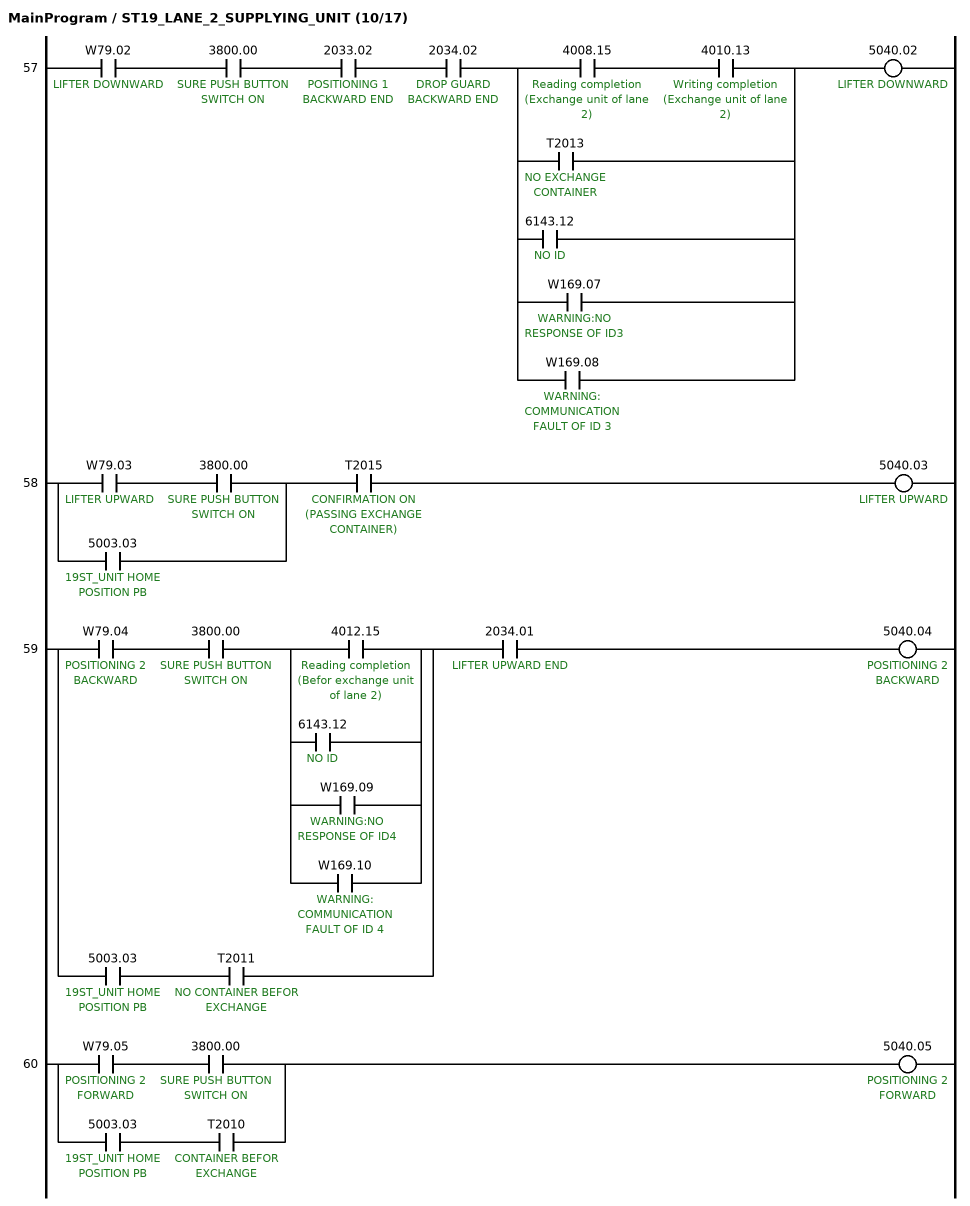
; [picture p696: MainProgram / ST19_LANE_2_SUPPLYING_UNIT, rungs 57-60]
; rung 57
LD W79.02  ; LIFTER DOWNWARD
AND 3800.00  ; SURE PUSH BUTTON SWITCH ON
AND 2033.02  ; POSITIONING 1 BACKWARD END
AND 2034.02  ; DROP GUARD BACKWARD END
LD 4008.15  ; Reading completion (Exchange unit of lane 2)
AND 4010.13  ; Writing completion (Exchange unit of lane 2)
OR T2013  ; NO EXCHANGE CONTAINER
OR 6143.12  ; NO ID
OR W169.07  ; WARNING:NO RESPONSE OF ID3
OR W169.08  ; WARNING:COMMUNICATION FAULT OF ID 3
ANDLD
OUT 5040.02  ; LIFTER DOWNWARD
; rung 58
LD W79.03  ; LIFTER UPWARD
AND 3800.00  ; SURE PUSH BUTTON SWITCH ON
OR 5003.03  ; 19ST_UNIT HOME POSITION PB
AND T2015  ; CONFIRMATION ON (PASSING EXCHANGE CONTAINER)
OUT 5040.03  ; LIFTER UPWARD
; rung 59
LD W79.04  ; POSITIONING 2 BACKWARD
AND 3800.00  ; SURE PUSH BUTTON SWITCH ON
LD 4012.15  ; Reading completion (Befor exchange unit of lane 2)
OR 6143.12  ; NO ID
OR W169.09  ; WARNING:NO RESPONSE OF ID4
OR W169.10  ; WARNING:COMMUNICATION FAULT OF ID 4
ANDLD
LD 5003.03  ; 19ST_UNIT HOME POSITION PB
AND T2011  ; NO CONTAINER BEFOR EXCHANGE
ORLD
AND 2034.01  ; LIFTER UPWARD END
OUT 5040.04  ; POSITIONING 2 BACKWARD
; rung 60
LD W79.05  ; POSITIONING 2 FORWARD
AND 3800.00  ; SURE PUSH BUTTON SWITCH ON
LD 5003.03  ; 19ST_UNIT HOME POSITION PB
AND T2010  ; CONTAINER BEFOR EXCHANGE
ORLD
OUT 5040.05  ; POSITIONING 2 FORWARD

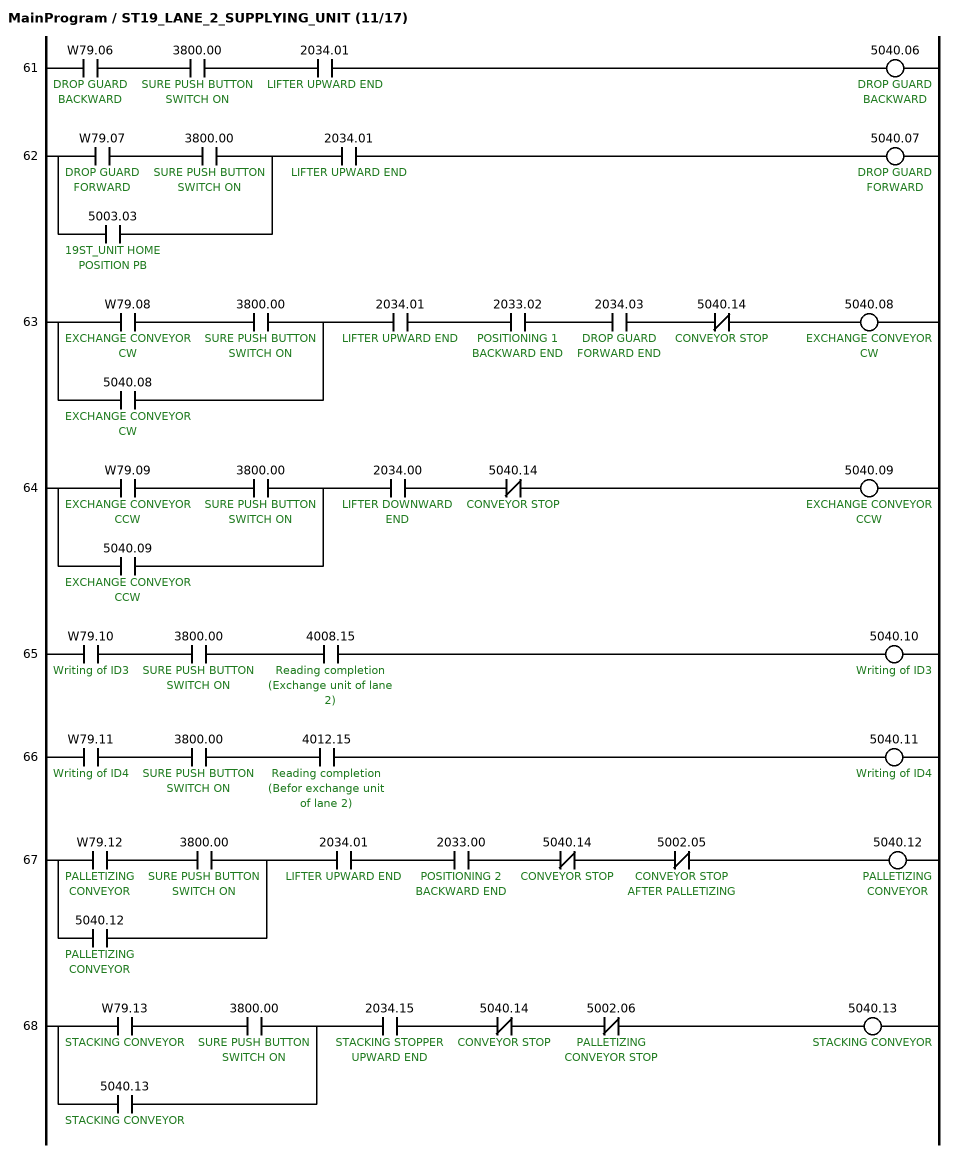
; rung 61
LD W79.06  ; DROP GUARD BACKWARD
AND 3800.00  ; SURE PUSH BUTTON SWITCH ON
AND 2034.01  ; LIFTER UPWARD END
OUT 5040.06  ; DROP GUARD BACKWARD
; rung 62
LD W79.07  ; DROP GUARD FORWARD
AND 3800.00  ; SURE PUSH BUTTON SWITCH ON
OR 5003.03  ; 19ST_UNIT HOME POSITION PB
AND 2034.01  ; LIFTER UPWARD END
OUT 5040.07  ; DROP GUARD FORWARD
; rung 63
LD W79.08  ; EXCHANGE CONVEYOR CW
AND 3800.00  ; SURE PUSH BUTTON SWITCH ON
OR 5040.08  ; EXCHANGE CONVEYOR CW
AND 2034.01  ; LIFTER UPWARD END
AND 2033.02  ; POSITIONING 1 BACKWARD END
AND 2034.03  ; DROP GUARD FORWARD END
ANDNOT 5040.14  ; CONVEYOR STOP
OUT 5040.08  ; EXCHANGE CONVEYOR CW
; rung 64
LD W79.09  ; EXCHANGE CONVEYOR CCW
AND 3800.00  ; SURE PUSH BUTTON SWITCH ON
OR 5040.09  ; EXCHANGE CONVEYOR CCW
AND 2034.00  ; LIFTER DOWNWARD END
ANDNOT 5040.14  ; CONVEYOR STOP
OUT 5040.09  ; EXCHANGE CONVEYOR CCW
; rung 65
LD W79.10  ; Writing of ID3
AND 3800.00  ; SURE PUSH BUTTON SWITCH ON
AND 4008.15  ; Reading completion (Exchange unit of lane 2)
OUT 5040.10  ; Writing of ID3
; rung 66
LD W79.11  ; Writing of ID4
AND 3800.00  ; SURE PUSH BUTTON SWITCH ON
AND 4012.15  ; Reading completion (Befor exchange unit of lane 2)
OUT 5040.11  ; Writing of ID4
; rung 67
LD W79.12  ; PALLETIZING CONVEYOR
AND 3800.00  ; SURE PUSH BUTTON SWITCH ON
OR 5040.12  ; PALLETIZING CONVEYOR
AND 2034.01  ; LIFTER UPWARD END
AND 2033.00  ; POSITIONING 2 BACKWARD END
ANDNOT 5040.14  ; CONVEYOR STOP
ANDNOT 5002.05  ; CONVEYOR STOP AFTER PALLETIZING
OUT 5040.12  ; PALLETIZING CONVEYOR
; rung 68
LD W79.13  ; STACKING CONVEYOR
AND 3800.00  ; SURE PUSH BUTTON SWITCH ON
OR 5040.13  ; STACKING CONVEYOR
AND 2034.15  ; STACKING STOPPER UPWARD END
ANDNOT 5040.14  ; CONVEYOR STOP
ANDNOT 5002.06  ; PALLETIZING CONVEYOR STOP
OUT 5040.13  ; STACKING CONVEYOR

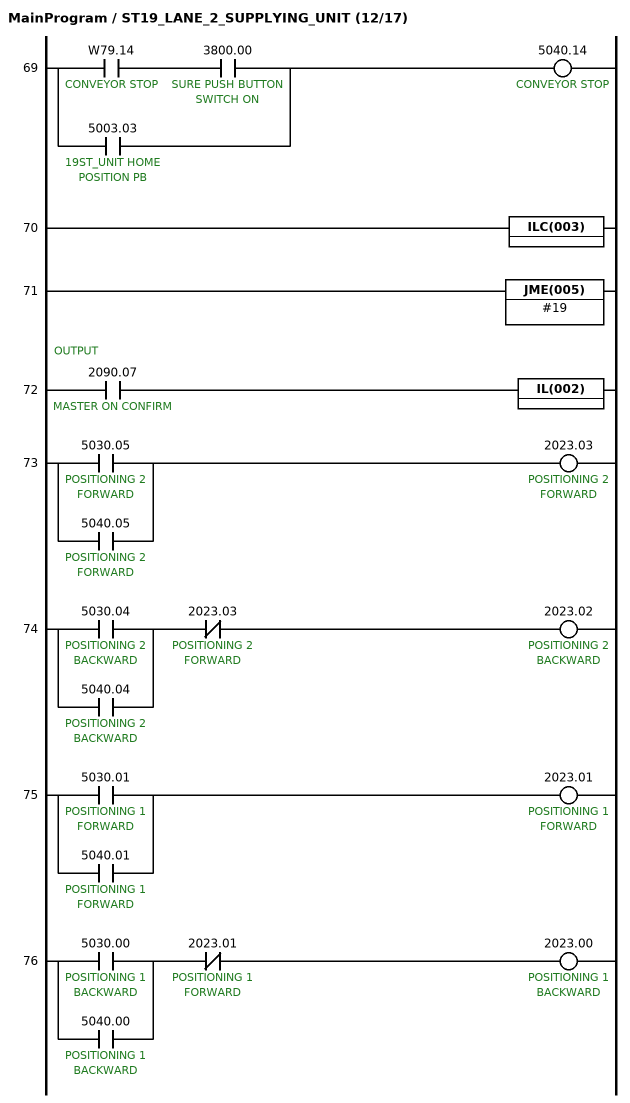
; rung 69
LD W79.14  ; CONVEYOR STOP
AND 3800.00  ; SURE PUSH BUTTON SWITCH ON
OR 5003.03  ; 19ST_UNIT HOME POSITION PB
OUT 5040.14  ; CONVEYOR STOP
; rung 70
ILC(003)
; rung 71
JME(005) #19
; rung 72: OUTPUT
LD 2090.07  ; MASTER ON CONFIRM
IL(002)
; rung 73
LD 5030.05  ; POSITIONING 2 FORWARD
OR 5040.05  ; POSITIONING 2 FORWARD
OUT 2023.03  ; POSITIONING 2 FORWARD
; rung 74
LD 5030.04  ; POSITIONING 2 BACKWARD
OR 5040.04  ; POSITIONING 2 BACKWARD
ANDNOT 2023.03  ; POSITIONING 2 FORWARD
OUT 2023.02  ; POSITIONING 2 BACKWARD
; rung 75
LD 5030.01  ; POSITIONING 1 FORWARD
OR 5040.01  ; POSITIONING 1 FORWARD
OUT 2023.01  ; POSITIONING 1 FORWARD
; rung 76
LD 5030.00  ; POSITIONING 1 BACKWARD
OR 5040.00  ; POSITIONING 1 BACKWARD
ANDNOT 2023.01  ; POSITIONING 1 FORWARD
OUT 2023.00  ; POSITIONING 1 BACKWARD

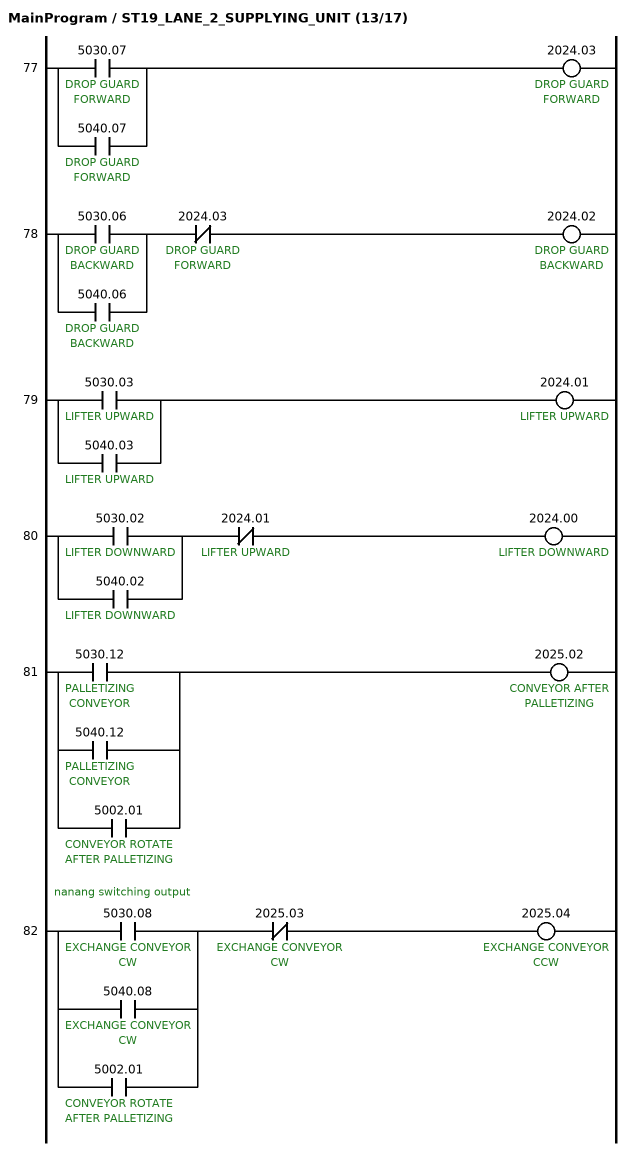
; rung 77
LD 5030.07  ; DROP GUARD FORWARD
OR 5040.07  ; DROP GUARD FORWARD
OUT 2024.03  ; DROP GUARD FORWARD
; rung 78
LD 5030.06  ; DROP GUARD BACKWARD
OR 5040.06  ; DROP GUARD BACKWARD
ANDNOT 2024.03  ; DROP GUARD FORWARD
OUT 2024.02  ; DROP GUARD BACKWARD
; rung 79
LD 5030.03  ; LIFTER UPWARD
OR 5040.03  ; LIFTER UPWARD
OUT 2024.01  ; LIFTER UPWARD
; rung 80
LD 5030.02  ; LIFTER DOWNWARD
OR 5040.02  ; LIFTER DOWNWARD
ANDNOT 2024.01  ; LIFTER UPWARD
OUT 2024.00  ; LIFTER DOWNWARD
; rung 81
LD 5030.12  ; PALLETIZING CONVEYOR
OR 5040.12  ; PALLETIZING CONVEYOR
OR 5002.01  ; CONVEYOR ROTATE AFTER PALLETIZING
OUT 2025.02  ; CONVEYOR AFTER PALLETIZING
; rung 82: nanang switching output
LD 5030.08  ; EXCHANGE CONVEYOR CW
OR 5040.08  ; EXCHANGE CONVEYOR CW
OR 5002.01  ; CONVEYOR ROTATE AFTER PALLETIZING
ANDNOT 2025.03  ; EXCHANGE CONVEYOR CW
OUT 2025.04  ; EXCHANGE CONVEYOR CCW

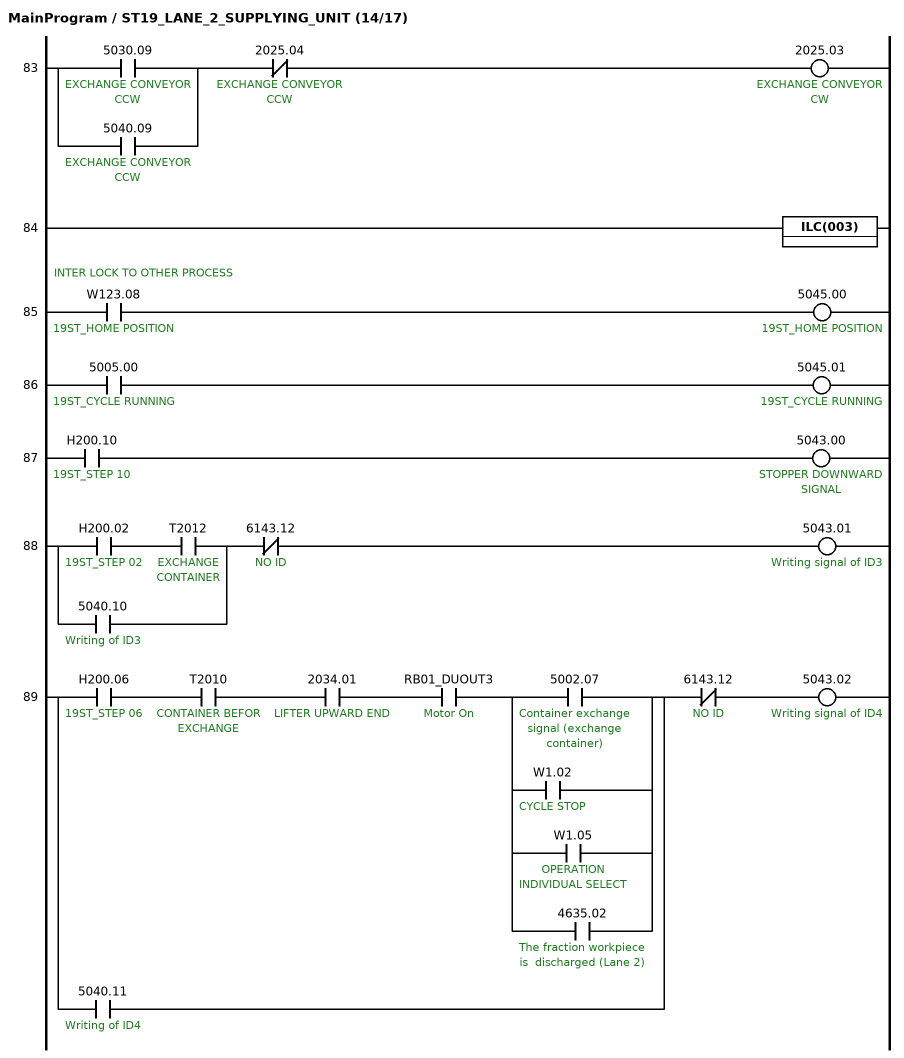
; rung 83
LD 5030.09  ; EXCHANGE CONVEYOR CCW
OR 5040.09  ; EXCHANGE CONVEYOR CCW
ANDNOT 2025.04  ; EXCHANGE CONVEYOR CCW
OUT 2025.03  ; EXCHANGE CONVEYOR CW
; rung 84
ILC(003)
; rung 85: INTER LOCK TO OTHER PROCESS
LD W123.08  ; 19ST_HOME POSITION
OUT 5045.00  ; 19ST_HOME POSITION
; rung 86
LD 5005.00  ; 19ST_CYCLE RUNNING
OUT 5045.01  ; 19ST_CYCLE RUNNING
; rung 87
LD H200.10  ; 19ST_STEP 10
OUT 5043.00  ; STOPPER DOWNWARD SIGNAL
; rung 88
LD H200.02  ; 19ST_STEP 02
AND T2012  ; EXCHANGE CONTAINER
OR 5040.10  ; Writing of ID3
ANDNOT 6143.12  ; NO ID
OUT 5043.01  ; Writing signal of ID3
; rung 89
LD H200.06  ; 19ST_STEP 06
AND T2010  ; CONTAINER BEFOR EXCHANGE
AND 2034.01  ; LIFTER UPWARD END
AND RB01_DUOUT3  ; Motor On
LD 5002.07  ; Container exchange signal (exchange container)
OR W1.02  ; CYCLE STOP
OR W1.05  ; OPERATION INDIVIDUAL SELECT
OR 4635.02  ; The fraction workpiece is  discharged (Lane 2)
ANDLD
OR 5040.11  ; Writing of ID4
ANDNOT 6143.12  ; NO ID
OUT 5043.02  ; Writing signal of ID4

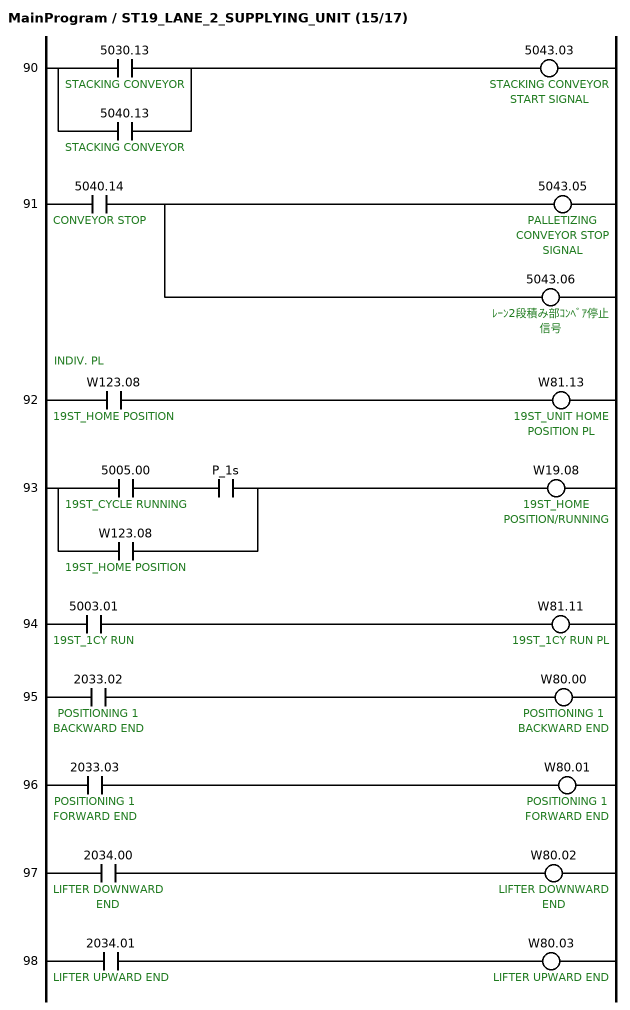
; rung 90
LD 5030.13  ; STACKING CONVEYOR
OR 5040.13  ; STACKING CONVEYOR
OUT 5043.03  ; STACKING CONVEYOR START SIGNAL
; rung 91
LD 5040.14  ; CONVEYOR STOP
OUT 5043.05  ; PALLETIZING CONVEYOR STOP SIGNAL
OUT 5043.06  ; ﾚｰﾝ2段積み部ｺﾝﾍﾞｱ停止信号
; rung 92: INDIV. PL
LD W123.08  ; 19ST_HOME POSITION
OUT W81.13  ; 19ST_UNIT HOME POSITION PL
; rung 93
LD 5005.00  ; 19ST_CYCLE RUNNING
AND P_1s
OR W123.08  ; 19ST_HOME POSITION
OUT W19.08  ; 19ST_HOME POSITION/RUNNING
; rung 94
LD 5003.01  ; 19ST_1CY RUN
OUT W81.11  ; 19ST_1CY RUN PL
; rung 95
LD 2033.02  ; POSITIONING 1 BACKWARD END
OUT W80.00  ; POSITIONING 1 BACKWARD END
; rung 96
LD 2033.03  ; POSITIONING 1 FORWARD END
OUT W80.01  ; POSITIONING 1 FORWARD END
; rung 97
LD 2034.00  ; LIFTER DOWNWARD END
OUT W80.02  ; LIFTER DOWNWARD END
; rung 98
LD 2034.01  ; LIFTER UPWARD END
OUT W80.03  ; LIFTER UPWARD END

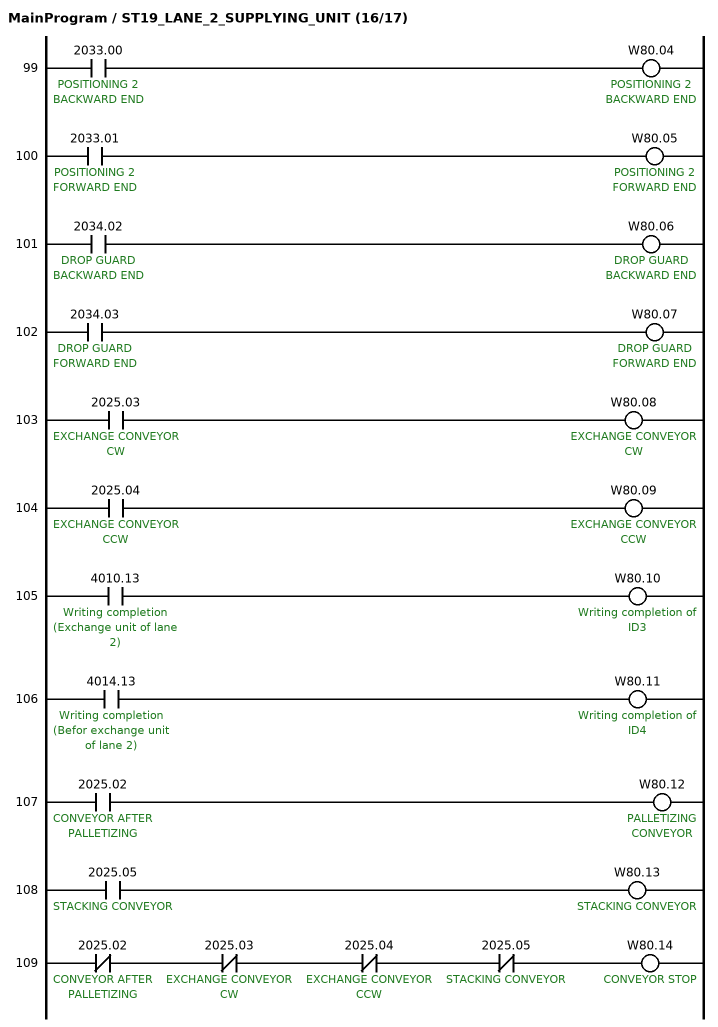
; rung 99
LD 2033.00  ; POSITIONING 2 BACKWARD END
OUT W80.04  ; POSITIONING 2 BACKWARD END
; rung 100
LD 2033.01  ; POSITIONING 2 FORWARD END
OUT W80.05  ; POSITIONING 2 FORWARD END
; rung 101
LD 2034.02  ; DROP GUARD BACKWARD END
OUT W80.06  ; DROP GUARD BACKWARD END
; rung 102
LD 2034.03  ; DROP GUARD FORWARD END
OUT W80.07  ; DROP GUARD FORWARD END
; rung 103
LD 2025.03  ; EXCHANGE CONVEYOR CW
OUT W80.08  ; EXCHANGE CONVEYOR CW
; rung 104
LD 2025.04  ; EXCHANGE CONVEYOR CCW
OUT W80.09  ; EXCHANGE CONVEYOR CCW
; rung 105
LD 4010.13  ; Writing completion (Exchange unit of lane 2)
OUT W80.10  ; Writing completion of ID3
; rung 106
LD 4014.13  ; Writing completion (Befor exchange unit of lane 2)
OUT W80.11  ; Writing completion of ID4
; rung 107
LD 2025.02  ; CONVEYOR AFTER PALLETIZING
OUT W80.12  ; PALLETIZING CONVEYOR
; rung 108
LD 2025.05  ; STACKING CONVEYOR
OUT W80.13  ; STACKING CONVEYOR
; rung 109
LDNOT 2025.02  ; CONVEYOR AFTER PALLETIZING
ANDNOT 2025.03  ; EXCHANGE CONVEYOR CW
ANDNOT 2025.04  ; EXCHANGE CONVEYOR CCW
ANDNOT 2025.05  ; STACKING CONVEYOR
OUT W80.14  ; CONVEYOR STOP

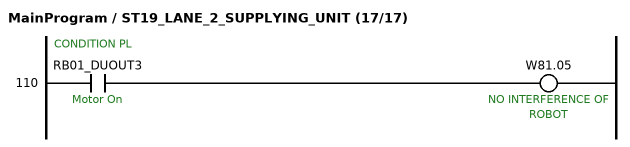
; rung 110: CONDITION PL
LD RB01_DUOUT3  ; Motor On
OUT W81.05  ; NO INTERFERENCE OF ROBOT

### Section ST20_LANE_2_STACKING_UNIT

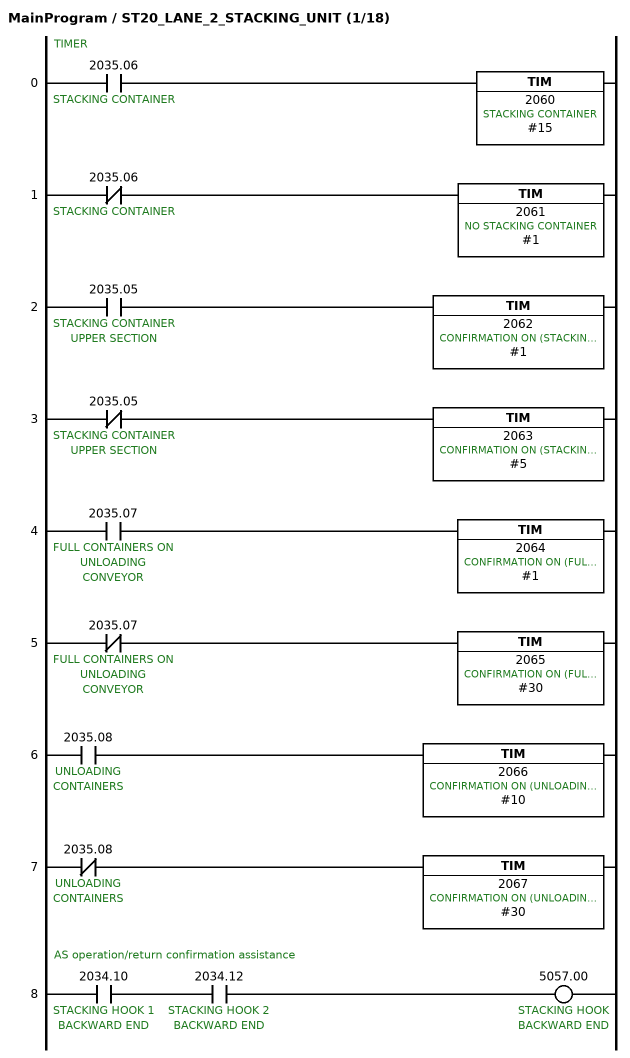
; rung 0: TIMER
LD 2035.06  ; STACKING CONTAINER
TIM 2060 #15  ; STACKING CONTAINER
; rung 1
LDNOT 2035.06  ; STACKING CONTAINER
TIM 2061 #1  ; NO STACKING CONTAINER
; rung 2
LD 2035.05  ; STACKING CONTAINER UPPER SECTION
TIM 2062 #1  ; CONFIRMATION ON (STACKING CONTAINER UPPER SECTION)
; rung 3
LDNOT 2035.05  ; STACKING CONTAINER UPPER SECTION
TIM 2063 #5  ; CONFIRMATION ON (STACKING CONTAINER UPPER SECTION)
; rung 4
LD 2035.07  ; FULL CONTAINERS ON UNLOADING CONVEYOR
TIM 2064 #1  ; CONFIRMATION ON (FULL CONTAINERS ON UNLOADING CONVEYOR)
; rung 5
LDNOT 2035.07  ; FULL CONTAINERS ON UNLOADING CONVEYOR
TIM 2065 #30  ; CONFIRMATION ON (FULL CONTAINERS ON UNLOADING CONVEYOR)
; rung 6
LD 2035.08  ; UNLOADING CONTAINERS
TIM 2066 #10  ; CONFIRMATION ON (UNLOADING CONTAINERS)
; rung 7
LDNOT 2035.08  ; UNLOADING CONTAINERS
TIM 2067 #30  ; CONFIRMATION ON (UNLOADING CONTAINERS)
; rung 8: AS operation/return confirmation assistance
LD 2034.10  ; STACKING HOOK 1 BACKWARD END
AND 2034.12  ; STACKING HOOK 2 BACKWARD END
OUT 5057.00  ; STACKING HOOK BACKWARD END

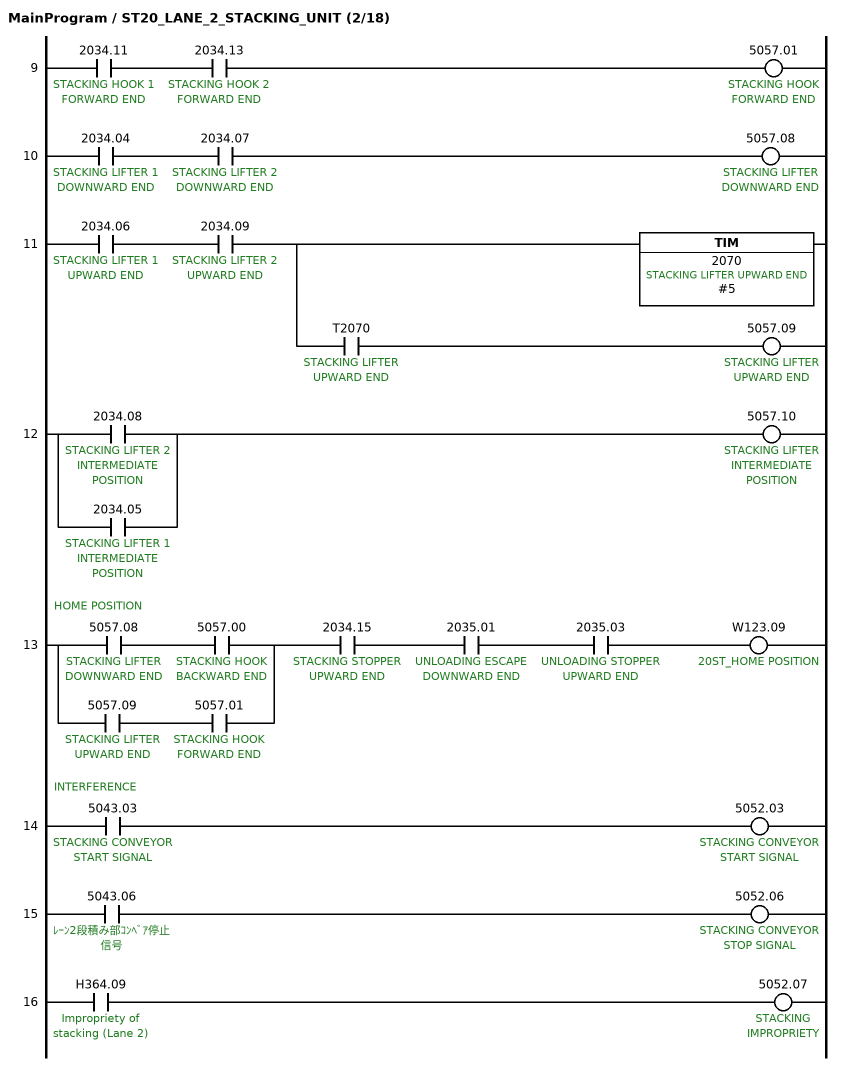
; rung 9
LD 2034.11  ; STACKING HOOK 1 FORWARD END
AND 2034.13  ; STACKING HOOK 2 FORWARD END
OUT 5057.01  ; STACKING HOOK FORWARD END
; rung 10
LD 2034.04  ; STACKING LIFTER 1 DOWNWARD END
AND 2034.07  ; STACKING LIFTER 2 DOWNWARD END
OUT 5057.08  ; STACKING LIFTER DOWNWARD END
; rung 11
LD 2034.06  ; STACKING LIFTER 1 UPWARD END
AND 2034.09  ; STACKING LIFTER 2 UPWARD END
TIM 2070 #5  ; STACKING LIFTER UPWARD END
AND T2070  ; STACKING LIFTER UPWARD END
OUT 5057.09  ; STACKING LIFTER UPWARD END
; rung 12
LD 2034.08  ; STACKING LIFTER 2 INTERMEDIATE POSITION
OR 2034.05  ; STACKING LIFTER 1 INTERMEDIATE POSITION
OUT 5057.10  ; STACKING LIFTER INTERMEDIATE POSITION
; rung 13: HOME POSITION
LD 5057.08  ; STACKING LIFTER DOWNWARD END
AND 5057.00  ; STACKING HOOK BACKWARD END
LD 5057.09  ; STACKING LIFTER UPWARD END
AND 5057.01  ; STACKING HOOK FORWARD END
ORLD
AND 2034.15  ; STACKING STOPPER UPWARD END
AND 2035.01  ; UNLOADING ESCAPE DOWNWARD END
AND 2035.03  ; UNLOADING STOPPER UPWARD END
OUT W123.09  ; 20ST_HOME POSITION
; rung 14: INTERFERENCE
LD 5043.03  ; STACKING CONVEYOR START SIGNAL
OUT 5052.03  ; STACKING CONVEYOR START SIGNAL
; rung 15
LD 5043.06  ; ﾚｰﾝ2段積み部ｺﾝﾍﾞｱ停止信号
OUT 5052.06  ; STACKING CONVEYOR STOP SIGNAL
; rung 16
LD H364.09  ; Impropriety of stacking (Lane 2)
OUT 5052.07  ; STACKING IMPROPRIETY

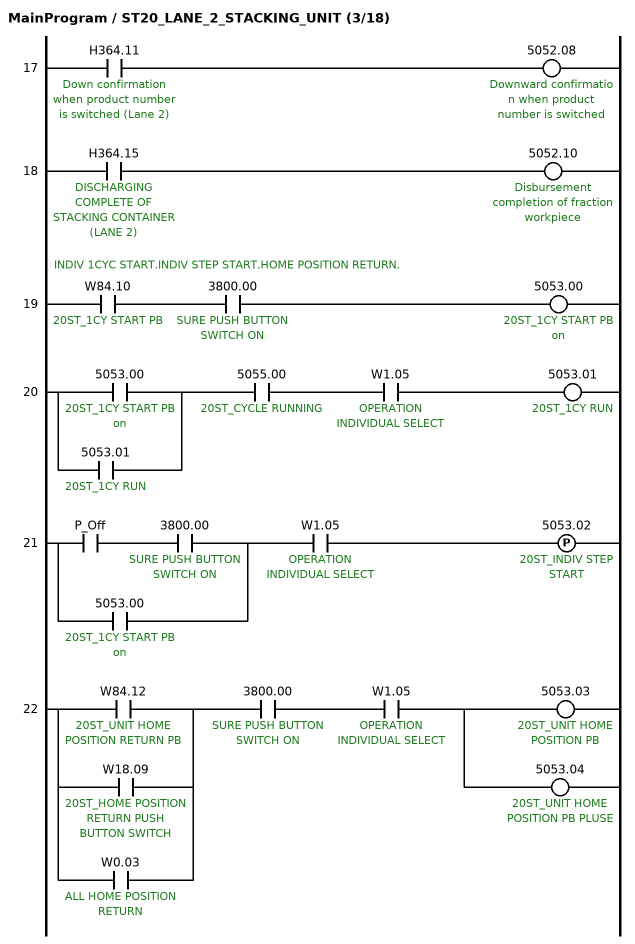
; rung 17
LD H364.11  ; Down confirmation when product number is switched (Lane 2)
OUT 5052.08  ; Downward confirmation when product number is switched
; rung 18
LD H364.15  ; DISCHARGING COMPLETE OF STACKING CONTAINER  (LANE 2)
OUT 5052.10  ; Disbursement completion of fraction workpiece
; rung 19: INDIV 1CYC START.INDIV STEP START.HOME POSITION RETURN.
LD W84.10  ; 20ST_1CY START PB
AND 3800.00  ; SURE PUSH BUTTON SWITCH ON
OUT 5053.00  ; 20ST_1CY START PB on
; rung 20
LD 5053.00  ; 20ST_1CY START PB on
OR 5053.01  ; 20ST_1CY RUN
AND 5055.00  ; 20ST_CYCLE RUNNING
AND W1.05  ; OPERATION INDIVIDUAL SELECT
OUT 5053.01  ; 20ST_1CY RUN
; rung 21
LD P_Off
AND 3800.00  ; SURE PUSH BUTTON SWITCH ON
OR 5053.00  ; 20ST_1CY START PB on
AND W1.05  ; OPERATION INDIVIDUAL SELECT
DIFU(013) 5053.02  ; 20ST_INDIV STEP START
; rung 22
LD W84.12  ; 20ST_UNIT HOME POSITION RETURN PB
OR W18.09  ; 20ST_HOME POSITION RETURN PUSH BUTTON SWITCH
OR W0.03  ; ALL HOME POSITION RETURN
AND 3800.00  ; SURE PUSH BUTTON SWITCH ON
AND W1.05  ; OPERATION INDIVIDUAL SELECT
OUT 5053.03  ; 20ST_UNIT HOME POSITION PB
OUT 5053.04  ; 20ST_UNIT HOME POSITION PB PLUSE

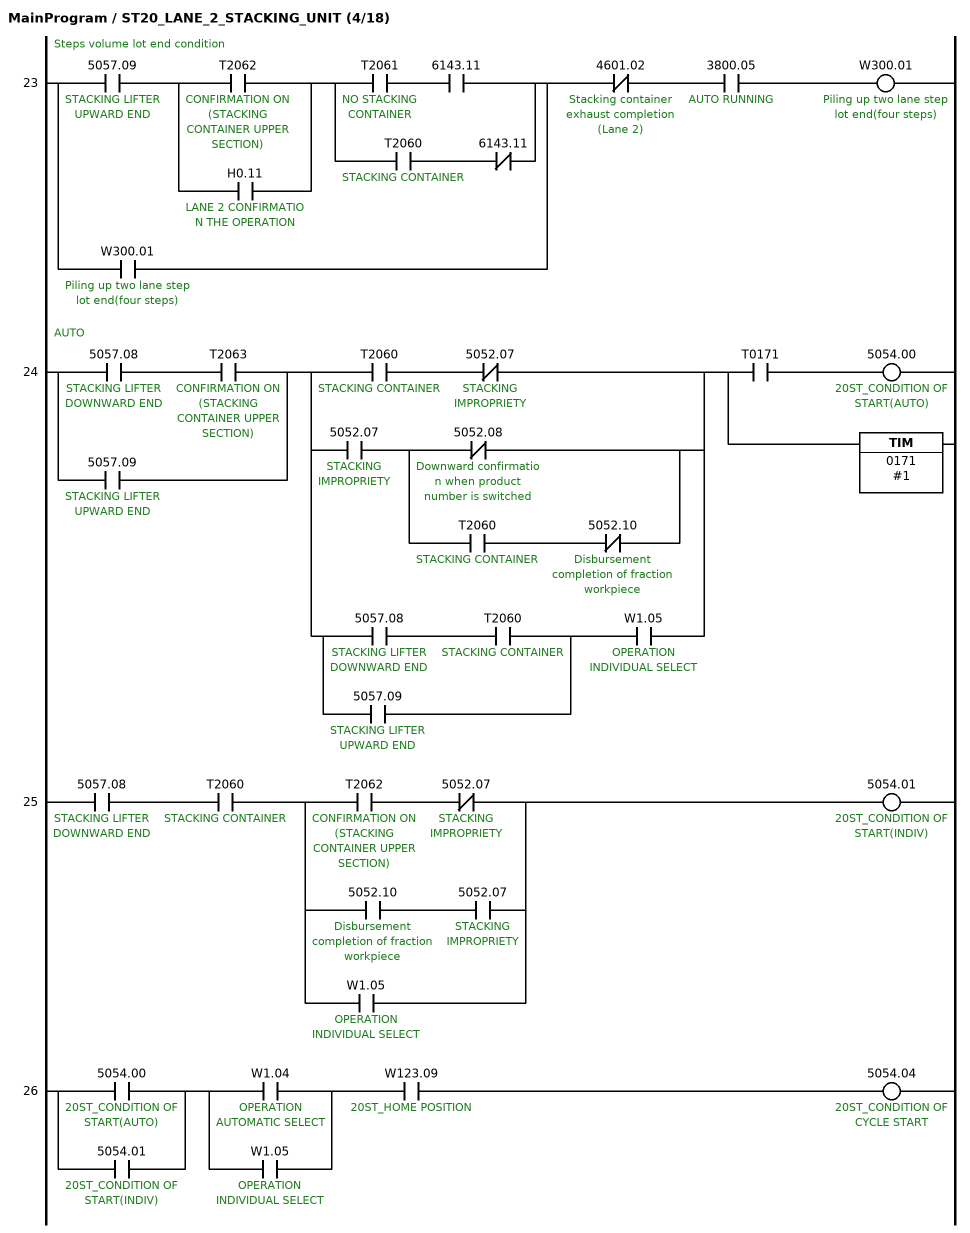
; rung 23: Steps volume lot end condition
LD 5057.09  ; STACKING LIFTER UPWARD END
LD T2062  ; CONFIRMATION ON (STACKING CONTAINER UPPER SECTION)
OR H0.11  ; LANE 2 CONFIRMATION THE OPERATION
ANDLD
LD T2061  ; NO STACKING CONTAINER
AND 6143.11
LD T2060  ; STACKING CONTAINER
ANDNOT 6143.11
ORLD
ANDLD
OR W300.01  ; Piling up two lane step lot end(four steps)
ANDNOT 4601.02  ; Stacking container exhaust completion (Lane 2)
AND 3800.05  ; AUTO RUNNING
OUT W300.01  ; Piling up two lane step lot end(four steps)
; rung 24: AUTO
LD 5057.08  ; STACKING LIFTER DOWNWARD END
AND T2063  ; CONFIRMATION ON (STACKING CONTAINER UPPER SECTION)
OR 5057.09  ; STACKING LIFTER UPWARD END
LD T2060  ; STACKING CONTAINER
ANDNOT 5052.07  ; STACKING IMPROPRIETY
LD 5052.07  ; STACKING IMPROPRIETY
LDNOT 5052.08  ; Downward confirmation when product number is switched
LD T2060  ; STACKING CONTAINER
ANDNOT 5052.10  ; Disbursement completion of fraction workpiece
ORLD
ANDLD
ORLD
LD 5057.08  ; STACKING LIFTER DOWNWARD END
AND T2060  ; STACKING CONTAINER
OR 5057.09  ; STACKING LIFTER UPWARD END
AND W1.05  ; OPERATION INDIVIDUAL SELECT
ORLD
ANDLD
OUT TR0
AND T0171
OUT 5054.00  ; 20ST_CONDITION OF START(AUTO)
LD TR0
TIM 0171 #1
; rung 25
LD 5057.08  ; STACKING LIFTER DOWNWARD END
AND T2060  ; STACKING CONTAINER
LD T2062  ; CONFIRMATION ON (STACKING CONTAINER UPPER SECTION)
ANDNOT 5052.07  ; STACKING IMPROPRIETY
LD 5052.10  ; Disbursement completion of fraction workpiece
AND 5052.07  ; STACKING IMPROPRIETY
ORLD
OR W1.05  ; OPERATION INDIVIDUAL SELECT
ANDLD
OUT 5054.01  ; 20ST_CONDITION OF START(INDIV)
; rung 26
LD 5054.00  ; 20ST_CONDITION OF START(AUTO)
OR 5054.01  ; 20ST_CONDITION OF START(INDIV)
LD W1.04  ; OPERATION AUTOMATIC SELECT
OR W1.05  ; OPERATION INDIVIDUAL SELECT
ANDLD
AND W123.09  ; 20ST_HOME POSITION
OUT 5054.04  ; 20ST_CONDITION OF CYCLE START

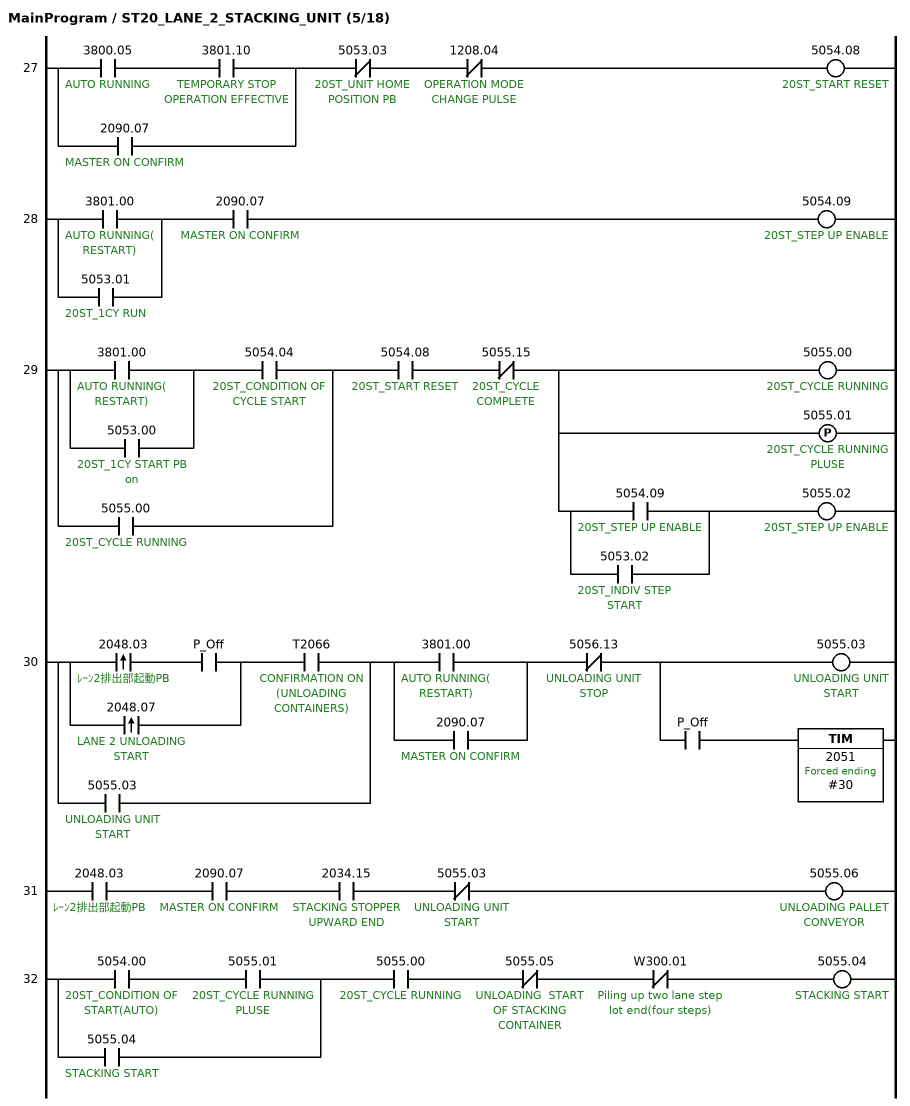
; rung 27
LD 3800.05  ; AUTO RUNNING
AND 3801.10  ; TEMPORARY STOP OPERATION EFFECTIVE
OR 2090.07  ; MASTER ON CONFIRM
ANDNOT 5053.03  ; 20ST_UNIT HOME POSITION PB
ANDNOT 1208.04  ; OPERATION MODE CHANGE PULSE
OUT 5054.08  ; 20ST_START RESET
; rung 28
LD 3801.00  ; AUTO RUNNING(RESTART)
OR 5053.01  ; 20ST_1CY RUN
AND 2090.07  ; MASTER ON CONFIRM
OUT 5054.09  ; 20ST_STEP UP ENABLE
; rung 29
LD 3801.00  ; AUTO RUNNING(RESTART)
OR 5053.00  ; 20ST_1CY START PB on
AND 5054.04  ; 20ST_CONDITION OF CYCLE START
OR 5055.00  ; 20ST_CYCLE RUNNING
AND 5054.08  ; 20ST_START RESET
ANDNOT 5055.15  ; 20ST_CYCLE COMPLETE
OUT 5055.00  ; 20ST_CYCLE RUNNING
DIFU(013) 5055.01  ; 20ST_CYCLE RUNNING PLUSE
LD 5054.09  ; 20ST_STEP UP ENABLE
OR 5053.02  ; 20ST_INDIV STEP START
ANDLD
OUT 5055.02  ; 20ST_STEP UP ENABLE
; rung 30
@LD 2048.03  ; ﾚｰﾝ2排出部起動PB
AND P_Off
@OR 2048.07  ; LANE 2 UNLOADING START
AND T2066  ; CONFIRMATION ON (UNLOADING CONTAINERS)
OR 5055.03  ; UNLOADING UNIT START
LD 3801.00  ; AUTO RUNNING(RESTART)
OR 2090.07  ; MASTER ON CONFIRM
ANDLD
ANDNOT 5056.13  ; UNLOADING UNIT STOP
OUT 5055.03  ; UNLOADING UNIT START
AND P_Off
TIM 2051 #30  ; Forced ending
; rung 31
LD 2048.03  ; ﾚｰﾝ2排出部起動PB
AND 2090.07  ; MASTER ON CONFIRM
AND 2034.15  ; STACKING STOPPER UPWARD END
ANDNOT 5055.03  ; UNLOADING UNIT START
OUT 5055.06  ; UNLOADING PALLET CONVEYOR
; rung 32
LD 5054.00  ; 20ST_CONDITION OF START(AUTO)
AND 5055.01  ; 20ST_CYCLE RUNNING PLUSE
OR 5055.04  ; STACKING START
AND 5055.00  ; 20ST_CYCLE RUNNING
ANDNOT 5055.05  ; UNLOADING  START OF STACKING CONTAINER
ANDNOT W300.01  ; Piling up two lane step lot end(four steps)
OUT 5055.04  ; STACKING START

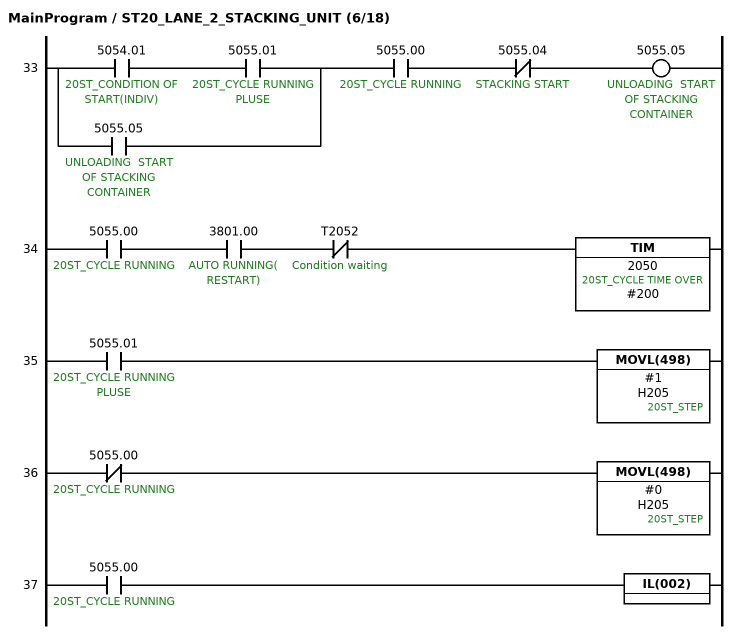
; rung 33
LD 5054.01  ; 20ST_CONDITION OF START(INDIV)
AND 5055.01  ; 20ST_CYCLE RUNNING PLUSE
OR 5055.05  ; UNLOADING  START OF STACKING CONTAINER
AND 5055.00  ; 20ST_CYCLE RUNNING
ANDNOT 5055.04  ; STACKING START
OUT 5055.05  ; UNLOADING  START OF STACKING CONTAINER
; rung 34
LD 5055.00  ; 20ST_CYCLE RUNNING
AND 3801.00  ; AUTO RUNNING(RESTART)
ANDNOT T2052  ; Condition waiting
TIM 2050 #200  ; 20ST_CYCLE TIME OVER
; rung 35
LD 5055.01  ; 20ST_CYCLE RUNNING PLUSE
MOVL(498) #1 H205  ; 20ST_STEP
; rung 36
LDNOT 5055.00  ; 20ST_CYCLE RUNNING
MOVL(498) #0 H205  ; 20ST_STEP
; rung 37
LD 5055.00  ; 20ST_CYCLE RUNNING
IL(002)

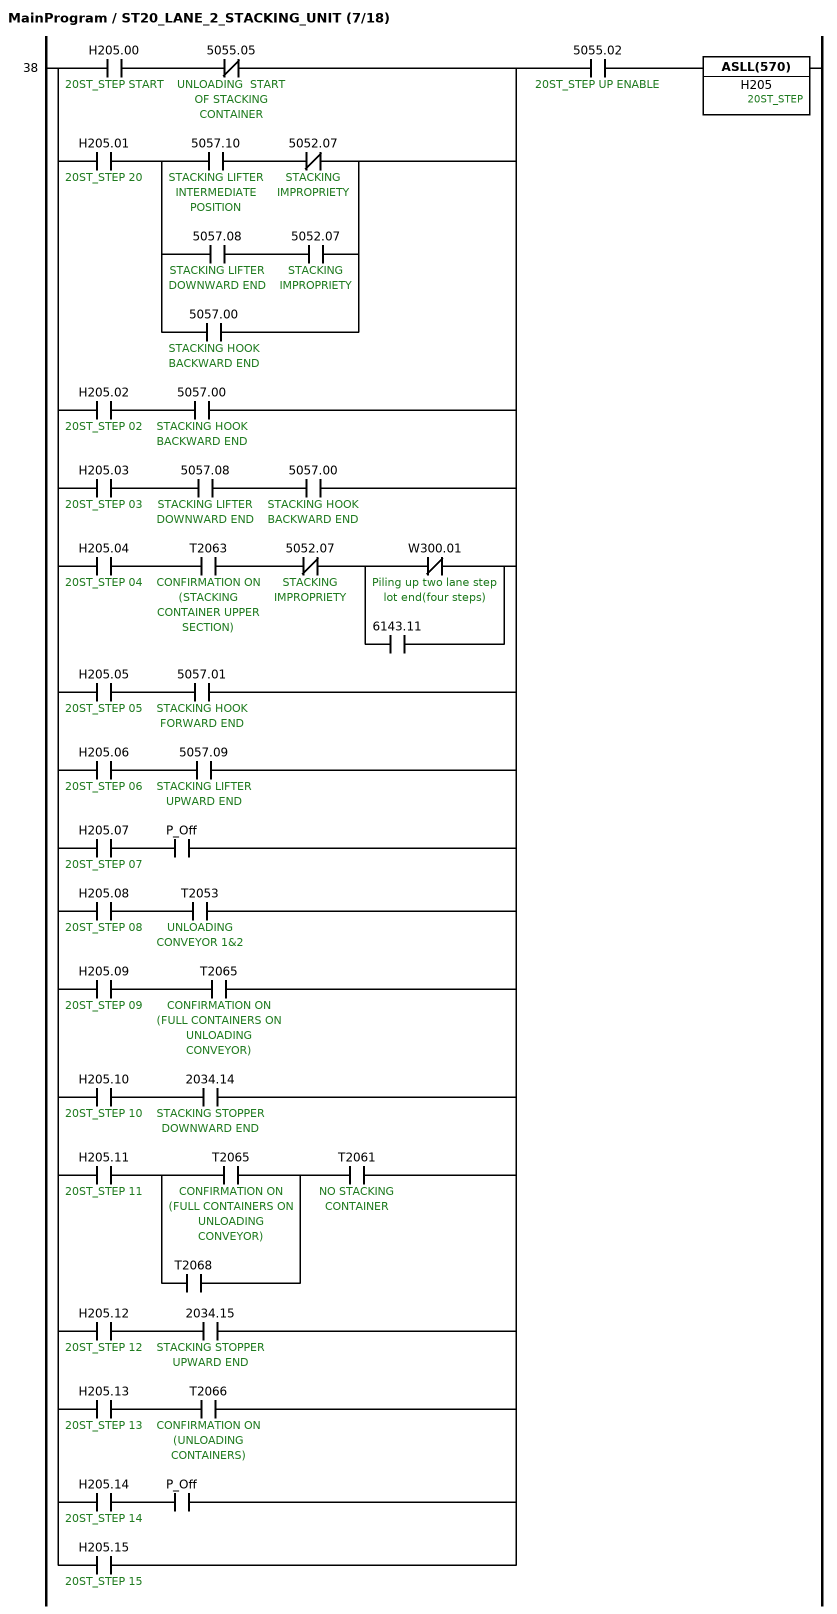
; rung 38
LD H205.00  ; 20ST_STEP START
ANDNOT 5055.05  ; UNLOADING  START OF STACKING CONTAINER
LD H205.01  ; 20ST_STEP 20
LD 5057.10  ; STACKING LIFTER INTERMEDIATE POSITION
ANDNOT 5052.07  ; STACKING IMPROPRIETY
LD 5057.08  ; STACKING LIFTER DOWNWARD END
AND 5052.07  ; STACKING IMPROPRIETY
ORLD
OR 5057.00  ; STACKING HOOK BACKWARD END
ANDLD
ORLD
LD H205.02  ; 20ST_STEP 02
AND 5057.00  ; STACKING HOOK BACKWARD END
ORLD
LD H205.03  ; 20ST_STEP 03
AND 5057.08  ; STACKING LIFTER DOWNWARD END
AND 5057.00  ; STACKING HOOK BACKWARD END
ORLD
LD H205.04  ; 20ST_STEP 04
AND T2063  ; CONFIRMATION ON (STACKING CONTAINER UPPER SECTION)
ANDNOT 5052.07  ; STACKING IMPROPRIETY
LDNOT W300.01  ; Piling up two lane step lot end(four steps)
OR 6143.11
ANDLD
ORLD
LD H205.05  ; 20ST_STEP 05
AND 5057.01  ; STACKING HOOK FORWARD END
ORLD
LD H205.06  ; 20ST_STEP 06
AND 5057.09  ; STACKING LIFTER UPWARD END
ORLD
LD H205.07  ; 20ST_STEP 07
AND P_Off
ORLD
LD H205.08  ; 20ST_STEP 08
AND T2053  ; UNLOADING CONVEYOR 1&2
ORLD
LD H205.09  ; 20ST_STEP 09
AND T2065  ; CONFIRMATION ON (FULL CONTAINERS ON UNLOADING CONVEYOR)
ORLD
LD H205.10  ; 20ST_STEP 10
AND 2034.14  ; STACKING STOPPER DOWNWARD END
ORLD
LD H205.11  ; 20ST_STEP 11
LD T2065  ; CONFIRMATION ON (FULL CONTAINERS ON UNLOADING CONVEYOR)
OR T2068
ANDLD
AND T2061  ; NO STACKING CONTAINER
ORLD
LD H205.12  ; 20ST_STEP 12
AND 2034.15  ; STACKING STOPPER UPWARD END
ORLD
LD H205.13  ; 20ST_STEP 13
AND T2066  ; CONFIRMATION ON (UNLOADING CONTAINERS)
ORLD
LD H205.14  ; 20ST_STEP 14
AND P_Off
ORLD
OR H205.15  ; 20ST_STEP 15
AND 5055.02  ; 20ST_STEP UP ENABLE
ASLL(570) H205  ; 20ST_STEP

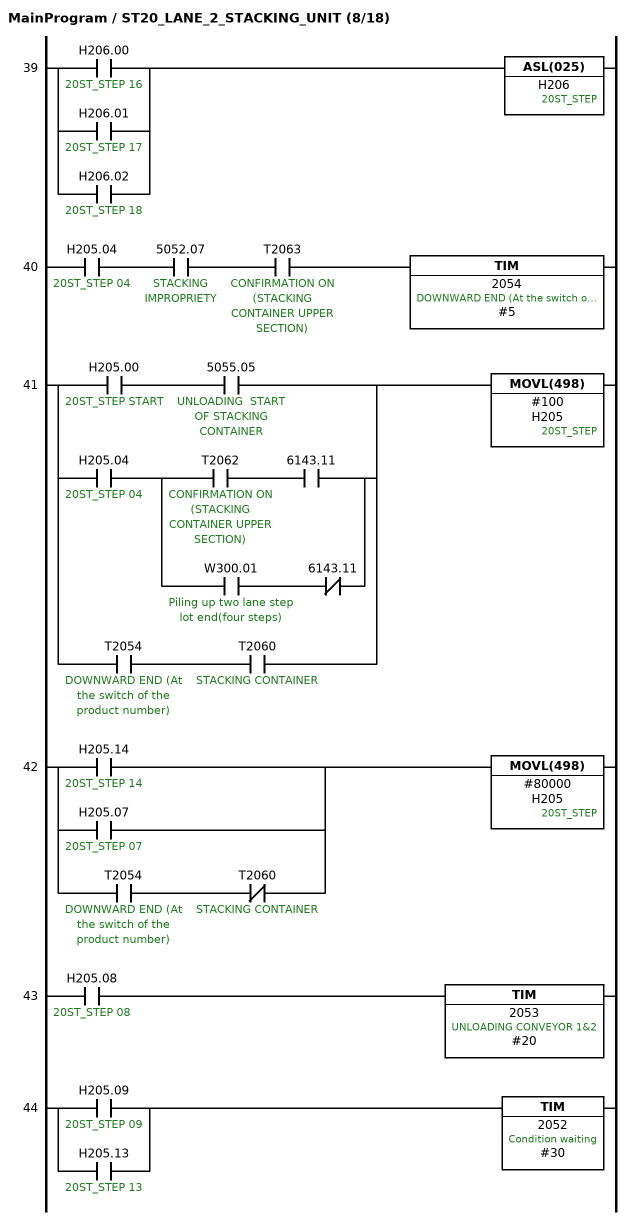
; rung 39
LD H206.00  ; 20ST_STEP 16
OR H206.01  ; 20ST_STEP 17
OR H206.02  ; 20ST_STEP 18
ASL(025) H206  ; 20ST_STEP
; rung 40
LD H205.04  ; 20ST_STEP 04
AND 5052.07  ; STACKING IMPROPRIETY
AND T2063  ; CONFIRMATION ON (STACKING CONTAINER UPPER SECTION)
TIM 2054 #5  ; DOWNWARD END (At the switch of the product number)
; rung 41
LD H205.00  ; 20ST_STEP START
AND 5055.05  ; UNLOADING  START OF STACKING CONTAINER
LD H205.04  ; 20ST_STEP 04
LD T2062  ; CONFIRMATION ON (STACKING CONTAINER UPPER SECTION)
AND 6143.11
LD W300.01  ; Piling up two lane step lot end(four steps)
ANDNOT 6143.11
ORLD
ANDLD
ORLD
LD T2054  ; DOWNWARD END (At the switch of the product number)
AND T2060  ; STACKING CONTAINER
ORLD
MOVL(498) #100 H205  ; 20ST_STEP
; rung 42
LD H205.14  ; 20ST_STEP 14
OR H205.07  ; 20ST_STEP 07
LD T2054  ; DOWNWARD END (At the switch of the product number)
ANDNOT T2060  ; STACKING CONTAINER
ORLD
MOVL(498) #80000 H205  ; 20ST_STEP
; rung 43
LD H205.08  ; 20ST_STEP 08
TIM 2053 #20  ; UNLOADING CONVEYOR 1&2
; rung 44
LD H205.09  ; 20ST_STEP 09
OR H205.13  ; 20ST_STEP 13
TIM 2052 #30  ; Condition waiting

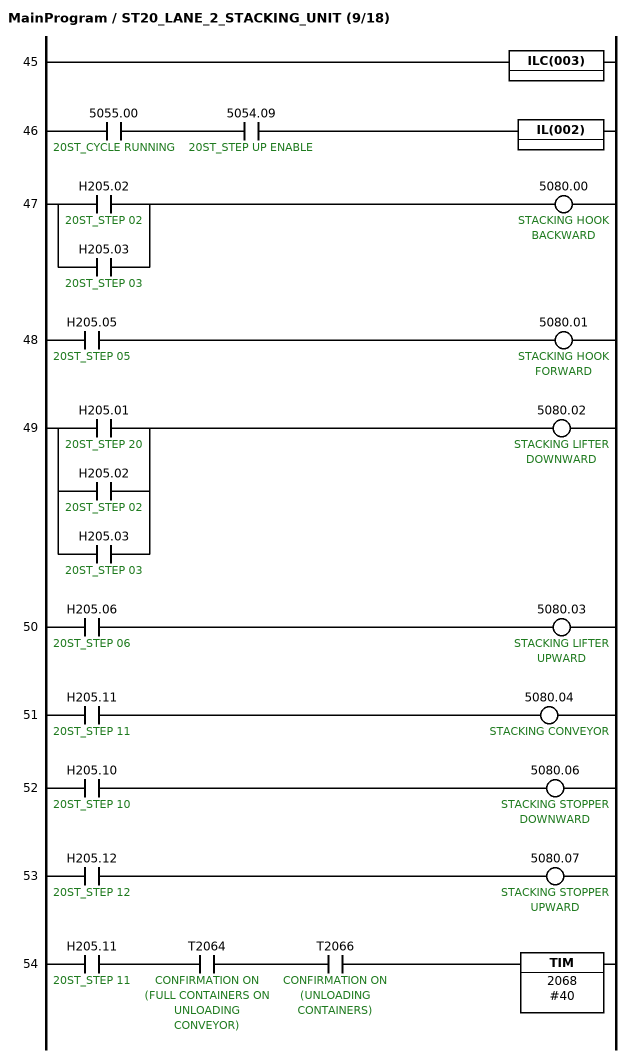
; rung 45
ILC(003)
; rung 46
LD 5055.00  ; 20ST_CYCLE RUNNING
AND 5054.09  ; 20ST_STEP UP ENABLE
IL(002)
; rung 47
LD H205.02  ; 20ST_STEP 02
OR H205.03  ; 20ST_STEP 03
OUT 5080.00  ; STACKING HOOK BACKWARD
; rung 48
LD H205.05  ; 20ST_STEP 05
OUT 5080.01  ; STACKING HOOK FORWARD
; rung 49
LD H205.01  ; 20ST_STEP 20
OR H205.02  ; 20ST_STEP 02
OR H205.03  ; 20ST_STEP 03
OUT 5080.02  ; STACKING LIFTER DOWNWARD
; rung 50
LD H205.06  ; 20ST_STEP 06
OUT 5080.03  ; STACKING LIFTER UPWARD
; rung 51
LD H205.11  ; 20ST_STEP 11
OUT 5080.04  ; STACKING CONVEYOR
; rung 52
LD H205.10  ; 20ST_STEP 10
OUT 5080.06  ; STACKING STOPPER DOWNWARD
; rung 53
LD H205.12  ; 20ST_STEP 12
OUT 5080.07  ; STACKING STOPPER UPWARD
; rung 54
LD H205.11  ; 20ST_STEP 11
AND T2064  ; CONFIRMATION ON (FULL CONTAINERS ON UNLOADING CONVEYOR)
AND T2066  ; CONFIRMATION ON (UNLOADING CONTAINERS)
TIM 2068 #40

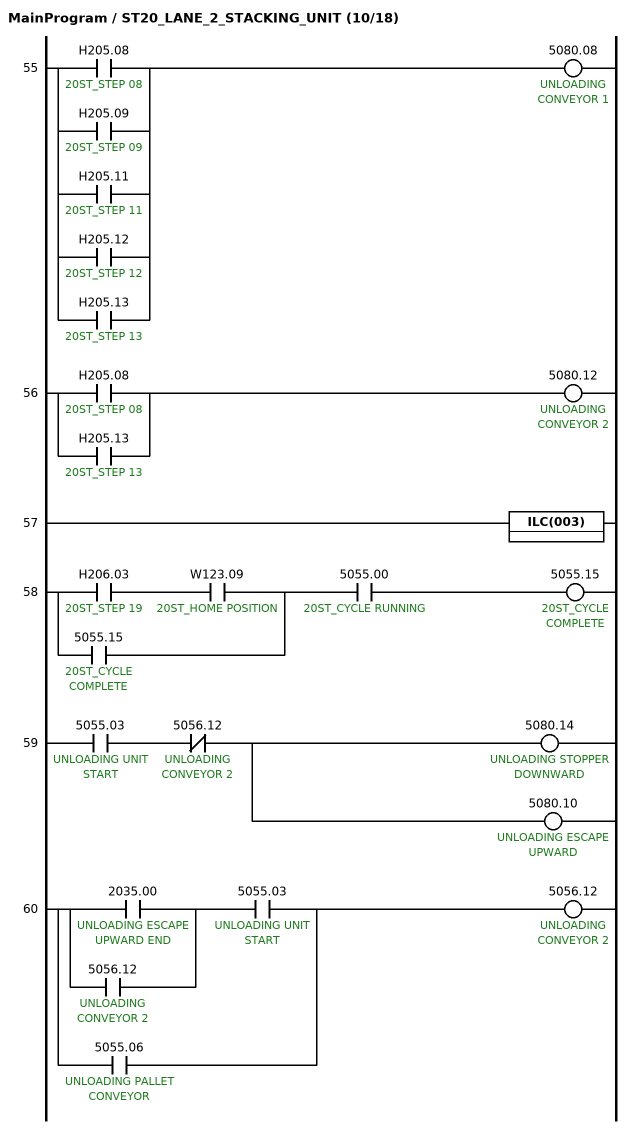
; rung 55
LD H205.08  ; 20ST_STEP 08
OR H205.09  ; 20ST_STEP 09
OR H205.11  ; 20ST_STEP 11
OR H205.12  ; 20ST_STEP 12
OR H205.13  ; 20ST_STEP 13
OUT 5080.08  ; UNLOADING CONVEYOR 1
; rung 56
LD H205.08  ; 20ST_STEP 08
OR H205.13  ; 20ST_STEP 13
OUT 5080.12  ; UNLOADING CONVEYOR 2
; rung 57
ILC(003)
; rung 58
LD H206.03  ; 20ST_STEP 19
AND W123.09  ; 20ST_HOME POSITION
OR 5055.15  ; 20ST_CYCLE COMPLETE
AND 5055.00  ; 20ST_CYCLE RUNNING
OUT 5055.15  ; 20ST_CYCLE COMPLETE
; rung 59
LD 5055.03  ; UNLOADING UNIT START
ANDNOT 5056.12  ; UNLOADING CONVEYOR 2
OUT 5080.14  ; UNLOADING STOPPER DOWNWARD
OUT 5080.10  ; UNLOADING ESCAPE UPWARD
; rung 60
LD 2035.00  ; UNLOADING ESCAPE UPWARD END
OR 5056.12  ; UNLOADING CONVEYOR 2
AND 5055.03  ; UNLOADING UNIT START
OR 5055.06  ; UNLOADING PALLET CONVEYOR
OUT 5056.12  ; UNLOADING CONVEYOR 2

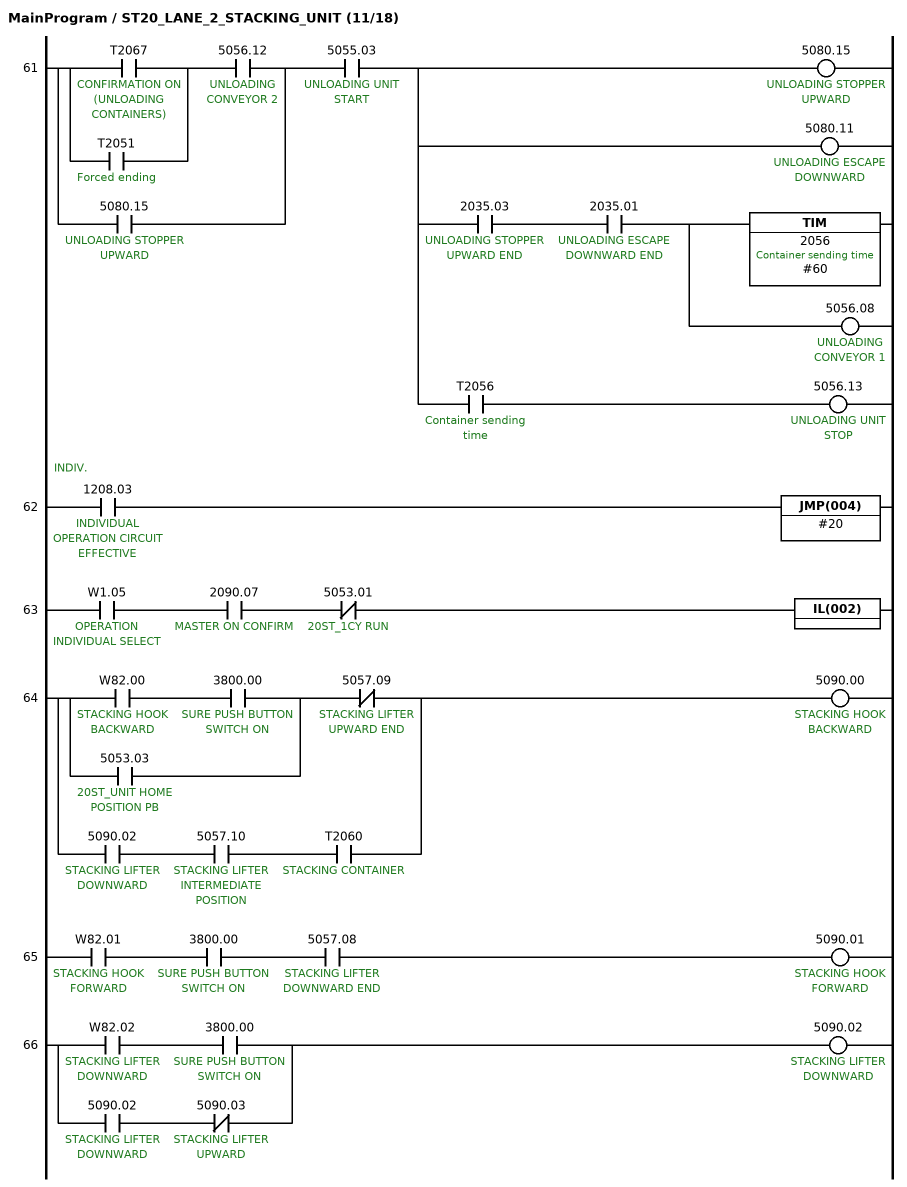
; rung 61
LD T2067  ; CONFIRMATION ON (UNLOADING CONTAINERS)
OR T2051  ; Forced ending
AND 5056.12  ; UNLOADING CONVEYOR 2
OR 5080.15  ; UNLOADING STOPPER UPWARD
AND 5055.03  ; UNLOADING UNIT START
OUT TR0
OUT 5080.15  ; UNLOADING STOPPER UPWARD
OUT 5080.11  ; UNLOADING ESCAPE DOWNWARD
AND 2035.03  ; UNLOADING STOPPER UPWARD END
AND 2035.01  ; UNLOADING ESCAPE DOWNWARD END
TIM 2056 #60  ; Container sending time
OUT 5056.08  ; UNLOADING CONVEYOR 1
LD TR0
AND T2056  ; Container sending time
OUT 5056.13  ; UNLOADING UNIT STOP
; rung 62: INDIV.
LD 1208.03  ; INDIVIDUAL OPERATION CIRCUIT EFFECTIVE
JMP(004) #20
; rung 63
LD W1.05  ; OPERATION INDIVIDUAL SELECT
AND 2090.07  ; MASTER ON CONFIRM
ANDNOT 5053.01  ; 20ST_1CY RUN
IL(002)
; rung 64
LD W82.00  ; STACKING HOOK BACKWARD
AND 3800.00  ; SURE PUSH BUTTON SWITCH ON
OR 5053.03  ; 20ST_UNIT HOME POSITION PB
ANDNOT 5057.09  ; STACKING LIFTER UPWARD END
LD 5090.02  ; STACKING LIFTER DOWNWARD
AND 5057.10  ; STACKING LIFTER INTERMEDIATE POSITION
AND T2060  ; STACKING CONTAINER
ORLD
OUT 5090.00  ; STACKING HOOK BACKWARD
; rung 65
LD W82.01  ; STACKING HOOK FORWARD
AND 3800.00  ; SURE PUSH BUTTON SWITCH ON
AND 5057.08  ; STACKING LIFTER DOWNWARD END
OUT 5090.01  ; STACKING HOOK FORWARD
; rung 66
LD W82.02  ; STACKING LIFTER DOWNWARD
AND 3800.00  ; SURE PUSH BUTTON SWITCH ON
LD 5090.02  ; STACKING LIFTER DOWNWARD
ANDNOT 5090.03  ; STACKING LIFTER UPWARD
ORLD
OUT 5090.02  ; STACKING LIFTER DOWNWARD

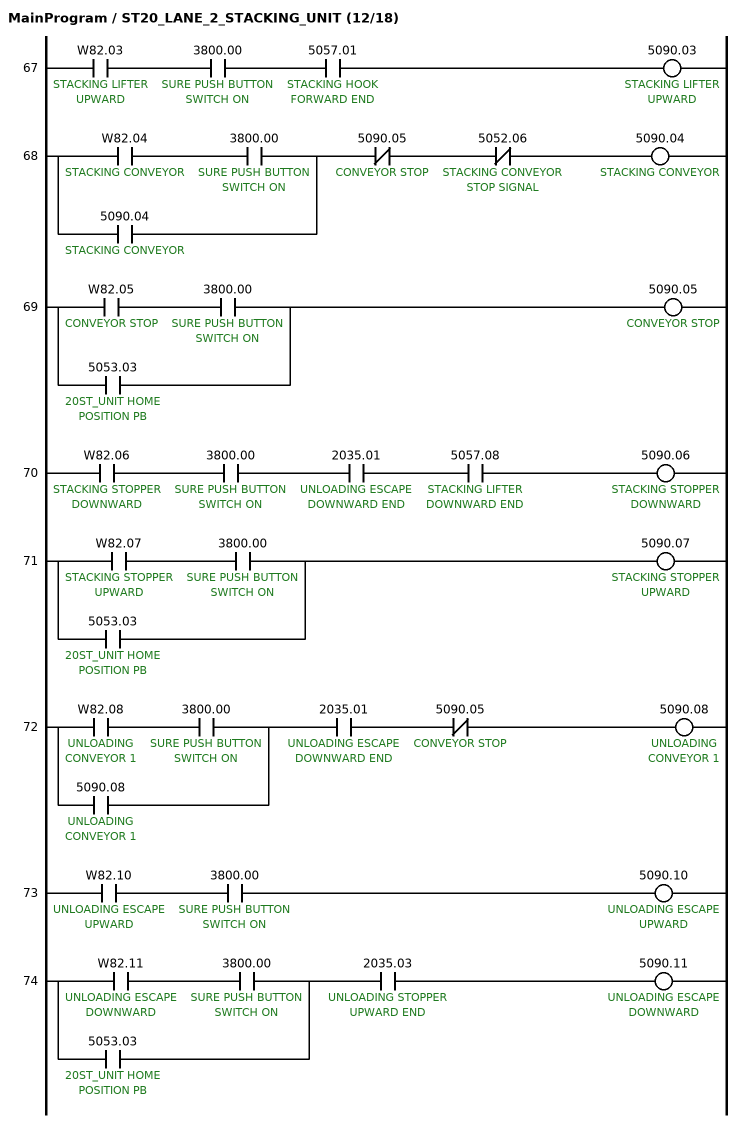
; rung 67
LD W82.03  ; STACKING LIFTER UPWARD
AND 3800.00  ; SURE PUSH BUTTON SWITCH ON
AND 5057.01  ; STACKING HOOK FORWARD END
OUT 5090.03  ; STACKING LIFTER UPWARD
; rung 68
LD W82.04  ; STACKING CONVEYOR
AND 3800.00  ; SURE PUSH BUTTON SWITCH ON
OR 5090.04  ; STACKING CONVEYOR
ANDNOT 5090.05  ; CONVEYOR STOP
ANDNOT 5052.06  ; STACKING CONVEYOR STOP SIGNAL
OUT 5090.04  ; STACKING CONVEYOR
; rung 69
LD W82.05  ; CONVEYOR STOP
AND 3800.00  ; SURE PUSH BUTTON SWITCH ON
OR 5053.03  ; 20ST_UNIT HOME POSITION PB
OUT 5090.05  ; CONVEYOR STOP
; rung 70
LD W82.06  ; STACKING STOPPER DOWNWARD
AND 3800.00  ; SURE PUSH BUTTON SWITCH ON
AND 2035.01  ; UNLOADING ESCAPE DOWNWARD END
AND 5057.08  ; STACKING LIFTER DOWNWARD END
OUT 5090.06  ; STACKING STOPPER DOWNWARD
; rung 71
LD W82.07  ; STACKING STOPPER UPWARD
AND 3800.00  ; SURE PUSH BUTTON SWITCH ON
OR 5053.03  ; 20ST_UNIT HOME POSITION PB
OUT 5090.07  ; STACKING STOPPER UPWARD
; rung 72
LD W82.08  ; UNLOADING CONVEYOR 1
AND 3800.00  ; SURE PUSH BUTTON SWITCH ON
OR 5090.08  ; UNLOADING CONVEYOR 1
AND 2035.01  ; UNLOADING ESCAPE DOWNWARD END
ANDNOT 5090.05  ; CONVEYOR STOP
OUT 5090.08  ; UNLOADING CONVEYOR 1
; rung 73
LD W82.10  ; UNLOADING ESCAPE UPWARD
AND 3800.00  ; SURE PUSH BUTTON SWITCH ON
OUT 5090.10  ; UNLOADING ESCAPE UPWARD
; rung 74
LD W82.11  ; UNLOADING ESCAPE DOWNWARD
AND 3800.00  ; SURE PUSH BUTTON SWITCH ON
OR 5053.03  ; 20ST_UNIT HOME POSITION PB
AND 2035.03  ; UNLOADING STOPPER UPWARD END
OUT 5090.11  ; UNLOADING ESCAPE DOWNWARD

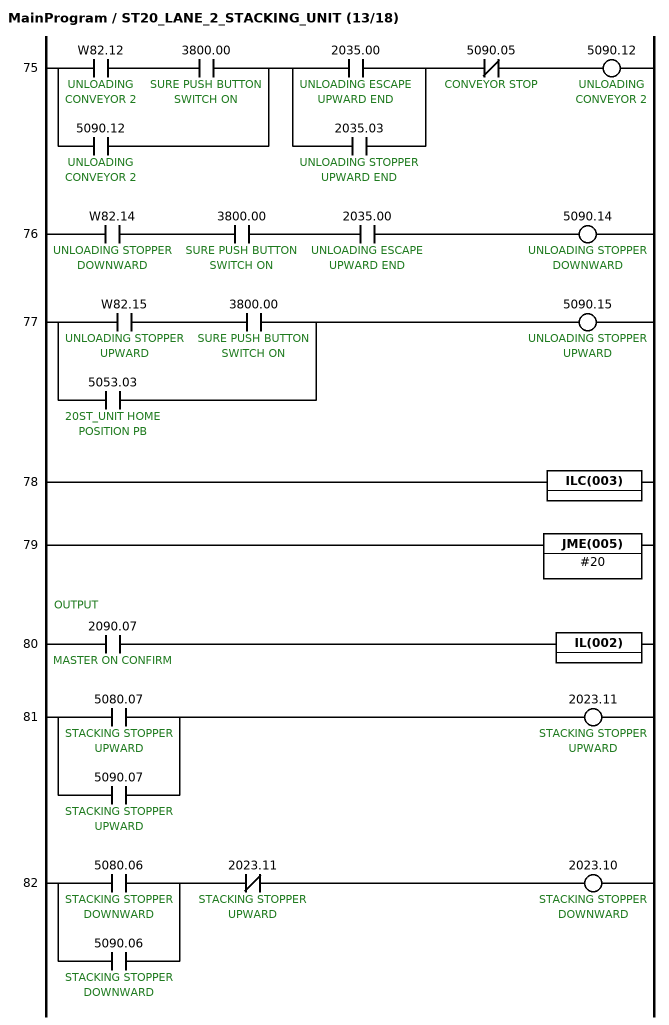
; rung 75
LD W82.12  ; UNLOADING CONVEYOR 2
AND 3800.00  ; SURE PUSH BUTTON SWITCH ON
OR 5090.12  ; UNLOADING CONVEYOR 2
LD 2035.00  ; UNLOADING ESCAPE UPWARD END
OR 2035.03  ; UNLOADING STOPPER UPWARD END
ANDLD
ANDNOT 5090.05  ; CONVEYOR STOP
OUT 5090.12  ; UNLOADING CONVEYOR 2
; rung 76
LD W82.14  ; UNLOADING STOPPER DOWNWARD
AND 3800.00  ; SURE PUSH BUTTON SWITCH ON
AND 2035.00  ; UNLOADING ESCAPE UPWARD END
OUT 5090.14  ; UNLOADING STOPPER DOWNWARD
; rung 77
LD W82.15  ; UNLOADING STOPPER UPWARD
AND 3800.00  ; SURE PUSH BUTTON SWITCH ON
OR 5053.03  ; 20ST_UNIT HOME POSITION PB
OUT 5090.15  ; UNLOADING STOPPER UPWARD
; rung 78
ILC(003)
; rung 79
JME(005) #20
; rung 80: OUTPUT
LD 2090.07  ; MASTER ON CONFIRM
IL(002)
; rung 81
LD 5080.07  ; STACKING STOPPER UPWARD
OR 5090.07  ; STACKING STOPPER UPWARD
OUT 2023.11  ; STACKING STOPPER UPWARD
; rung 82
LD 5080.06  ; STACKING STOPPER DOWNWARD
OR 5090.06  ; STACKING STOPPER DOWNWARD
ANDNOT 2023.11  ; STACKING STOPPER UPWARD
OUT 2023.10  ; STACKING STOPPER DOWNWARD

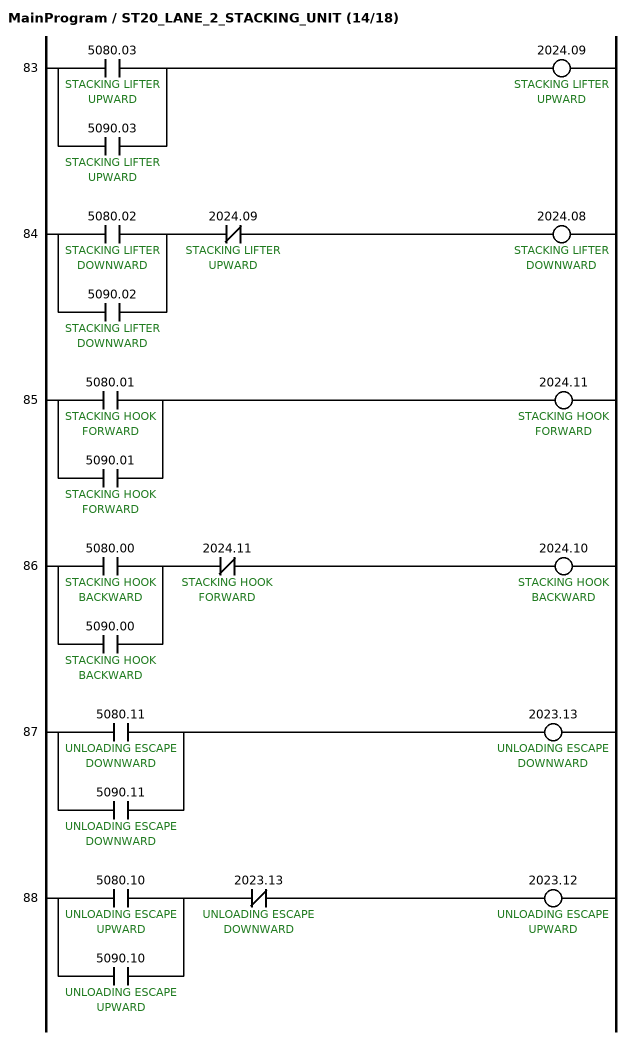
; rung 83
LD 5080.03  ; STACKING LIFTER UPWARD
OR 5090.03  ; STACKING LIFTER UPWARD
OUT 2024.09  ; STACKING LIFTER UPWARD
; rung 84
LD 5080.02  ; STACKING LIFTER DOWNWARD
OR 5090.02  ; STACKING LIFTER DOWNWARD
ANDNOT 2024.09  ; STACKING LIFTER UPWARD
OUT 2024.08  ; STACKING LIFTER DOWNWARD
; rung 85
LD 5080.01  ; STACKING HOOK FORWARD
OR 5090.01  ; STACKING HOOK FORWARD
OUT 2024.11  ; STACKING HOOK FORWARD
; rung 86
LD 5080.00  ; STACKING HOOK BACKWARD
OR 5090.00  ; STACKING HOOK BACKWARD
ANDNOT 2024.11  ; STACKING HOOK FORWARD
OUT 2024.10  ; STACKING HOOK BACKWARD
; rung 87
LD 5080.11  ; UNLOADING ESCAPE DOWNWARD
OR 5090.11  ; UNLOADING ESCAPE DOWNWARD
OUT 2023.13  ; UNLOADING ESCAPE DOWNWARD
; rung 88
LD 5080.10  ; UNLOADING ESCAPE UPWARD
OR 5090.10  ; UNLOADING ESCAPE UPWARD
ANDNOT 2023.13  ; UNLOADING ESCAPE DOWNWARD
OUT 2023.12  ; UNLOADING ESCAPE UPWARD

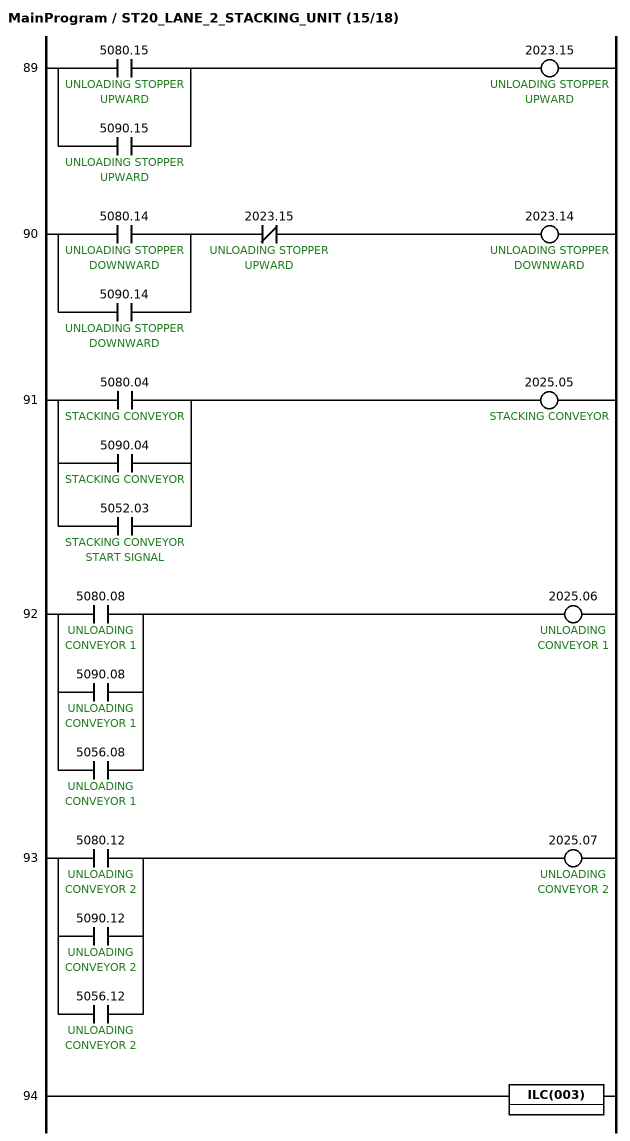
; rung 89
LD 5080.15  ; UNLOADING STOPPER UPWARD
OR 5090.15  ; UNLOADING STOPPER UPWARD
OUT 2023.15  ; UNLOADING STOPPER UPWARD
; rung 90
LD 5080.14  ; UNLOADING STOPPER DOWNWARD
OR 5090.14  ; UNLOADING STOPPER DOWNWARD
ANDNOT 2023.15  ; UNLOADING STOPPER UPWARD
OUT 2023.14  ; UNLOADING STOPPER DOWNWARD
; rung 91
LD 5080.04  ; STACKING CONVEYOR
OR 5090.04  ; STACKING CONVEYOR
OR 5052.03  ; STACKING CONVEYOR START SIGNAL
OUT 2025.05  ; STACKING CONVEYOR
; rung 92
LD 5080.08  ; UNLOADING CONVEYOR 1
OR 5090.08  ; UNLOADING CONVEYOR 1
OR 5056.08  ; UNLOADING CONVEYOR 1
OUT 2025.06  ; UNLOADING CONVEYOR 1
; rung 93
LD 5080.12  ; UNLOADING CONVEYOR 2
OR 5090.12  ; UNLOADING CONVEYOR 2
OR 5056.12  ; UNLOADING CONVEYOR 2
OUT 2025.07  ; UNLOADING CONVEYOR 2
; rung 94
ILC(003)

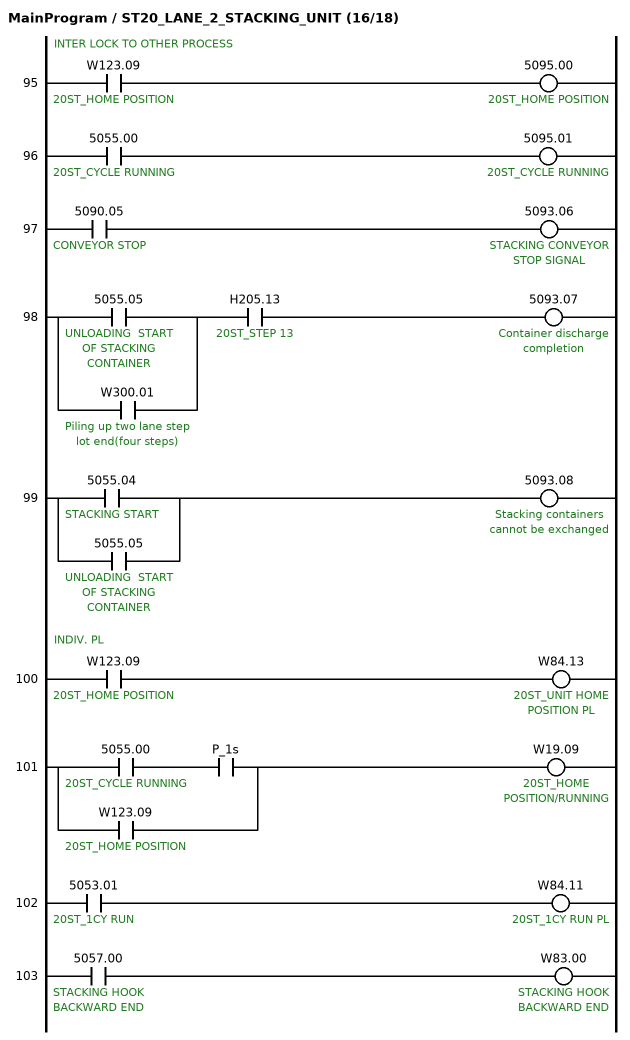
; rung 95: INTER LOCK TO OTHER PROCESS
LD W123.09  ; 20ST_HOME POSITION
OUT 5095.00  ; 20ST_HOME POSITION
; rung 96
LD 5055.00  ; 20ST_CYCLE RUNNING
OUT 5095.01  ; 20ST_CYCLE RUNNING
; rung 97
LD 5090.05  ; CONVEYOR STOP
OUT 5093.06  ; STACKING CONVEYOR STOP SIGNAL
; rung 98
LD 5055.05  ; UNLOADING  START OF STACKING CONTAINER
OR W300.01  ; Piling up two lane step lot end(four steps)
AND H205.13  ; 20ST_STEP 13
OUT 5093.07  ; Container discharge completion
; rung 99
LD 5055.04  ; STACKING START
OR 5055.05  ; UNLOADING  START OF STACKING CONTAINER
OUT 5093.08  ; Stacking containers cannot be exchanged
; rung 100: INDIV. PL
LD W123.09  ; 20ST_HOME POSITION
OUT W84.13  ; 20ST_UNIT HOME POSITION PL
; rung 101
LD 5055.00  ; 20ST_CYCLE RUNNING
AND P_1s
OR W123.09  ; 20ST_HOME POSITION
OUT W19.09  ; 20ST_HOME POSITION/RUNNING
; rung 102
LD 5053.01  ; 20ST_1CY RUN
OUT W84.11  ; 20ST_1CY RUN PL
; rung 103
LD 5057.00  ; STACKING HOOK BACKWARD END
OUT W83.00  ; STACKING HOOK BACKWARD END

